PROGRAM MAIN
VAR
	execute : BOOL;
	stop : BOOL;
	manualStep : BOOL := TRUE;
	manualSuction : BOOL;
	
	moduleWB : WoodBunkEx;
	moduleCIP : ChipboardEx;
	exec1, exec2 : BOOL;
END_VAR

CallHardware(); //start program with hardware call - pass values and arrays into function blocks
SetupHardware(); //initialize values

//callModules(); ST
runModules(); //LLD

CallHardware(); //end program with hardware call

ACTION callModules:
moduleWB(
	execute:= exec1, 
	stop:= stop, 
	manualStep:= manualStep, 
	manualSuction:= manualSuction,
 
	robotLeft:= robot1, 
	robotRight:= robot2, 
	toolStorageLeft:= toolStorageA21Left, 
	toolStorageRight:= toolStorageA21Right, 
	stagingTableLeft:= stagingTableLeft, 
	stagingTableRight:= stagingTableRight, 
	magazineLeft:= magazineA21Left, 
	magazineRight:= magazineA21Right, 
	strapper:= strapperA21, 
	horizontalDriveLeft:= horizontalDriveA21Left, 
	horizontalDriveRight:= horizontalDriveA21Right, 
	verticalDriveLeft:= verticalDriveA21Left, 
	verticalDriveRight:= verticalDriveA21Right, 
	pistonBottom:= pistonA21Bottom, 
	suctionTop:= suctionA21Top, 
	suctionLeft:= suctionA21Left, 
	suctionRight:= suctionA21Right, 
	suctionBottom:= suctionA21Bottom, 
	
	done=> ,
	generalError=> , 
	errorLeft=> , 
	errorRight=> );
	

moduleCIP(
	execute:= exec2, 
	stop:= stop, 
	manualStep:= manualStep, 
	
	robotLeft:= robot1, 
	robotRight:= robot2, 
	toolStorageLeft:= toolStorageA21Left, 
	toolStorageRight:= toolStorageA21Right,
	skidLeft:= skidA21Left, 
	skidRight:= skidA21Right, 
	
	done=> , 
	generalError=> , 
	failLeft=> , 
	failRight=> );
END_ACTION

ACTION runModules:
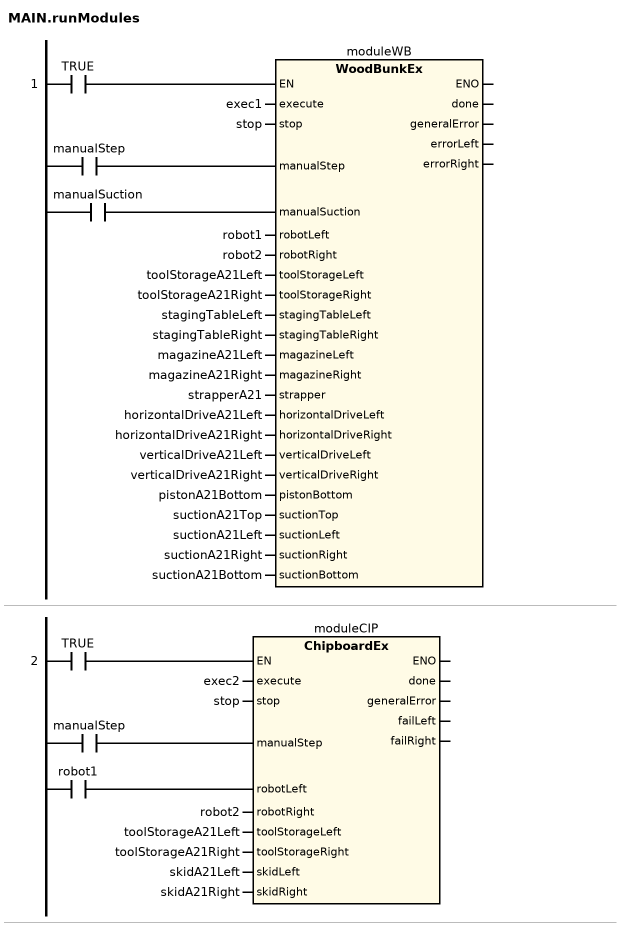
// NETWORK 1
moduleWB(
    execute := exec1,
    stop := stop,
    manualStep := manualStep,
    manualSuction := manualSuction,
    robotLeft := robot1,
    robotRight := robot2,
    toolStorageLeft := toolStorageA21Left,
    toolStorageRight := toolStorageA21Right,
    stagingTableLeft := stagingTableLeft,
    stagingTableRight := stagingTableRight,
    magazineLeft := magazineA21Left,
    magazineRight := magazineA21Right,
    strapper := strapperA21,
    horizontalDriveLeft := horizontalDriveA21Left,
    horizontalDriveRight := horizontalDriveA21Right,
    verticalDriveLeft := verticalDriveA21Left,
    verticalDriveRight := verticalDriveA21Right,
    pistonBottom := pistonA21Bottom,
    suctionTop := suctionA21Top,
    suctionLeft := suctionA21Left,
    suctionRight := suctionA21Right,
    suctionBottom := suctionA21Bottom); // WoodBunkEx

// NETWORK 2
moduleCIP(
    execute := exec2,
    stop := stop,
    manualStep := manualStep,
    robotLeft := robot1,
    robotRight := robot2,
    toolStorageLeft := toolStorageA21Left,
    toolStorageRight := toolStorageA21Right,
    skidLeft := skidA21Left,
    skidRight := skidA21Right); // ChipboardEx
END_ACTION

END_PROGRAM

(* stored: Version 1.1.0.1, ProductVersion 3.1.4024.11
   POU MAIN: Id {9caf58b7-eccf-4a65-a3e3-2c8d81beb312}, SpecialFunc None
   Action callModules: Id {3bfb8053-bd3a-41f1-92ca-bb3cb5200abe}
   Action runModules: Id {797c012e-5535-4cfd-a7fe-f38cfe08cb9f} *)
